TYPE "ValveMachine_PB"
VERSION : 0.1
// Block: ValveMachine_PB
   STRUCT
      Rest : Bool;
      Work : Bool;
      StartStop : Bool;
   END_STRUCT;

END_TYPE
